{attribute 'qualified_only'}
VAR_GLOBAL
	//	global vbariables
	
	RunStop			AT %Q*	: BOOL;
	ErrAck			AT %Q*	: BOOL;
	
	SafetyAndOut	AT %I*	: BOOL;
	
END_VAR

(* stored: Version 1.1.0.1, ProductVersion 3.1.4024.11
   GVL GVL: Id {0b7266af-4ab7-4dfb-8024-0b65739ab4c6} *)
